FUNCTION_BLOCK CylControl (* Basic Function Block Type *)
  (* Standard: 61499-2 *)
  (* Version 0.0, 8/12/2014, valvya, nxtControl GmbH, Template *)
  PACKAGE Main;
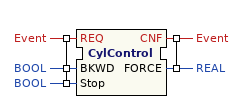
  EVENT_INPUT
    REQ WITH BKWD, Stop; (* Normal Execution Request *)
  END_EVENT
  EVENT_OUTPUT
    CNF WITH FORCE; (* Execution Confirmation *)
  END_EVENT
  VAR_INPUT
    BKWD : BOOL; (* Input event qualifier *)
    Stop : BOOL;
  END_VAR
  VAR_OUTPUT
    FORCE : REAL; (* Output event qualifier *)
  END_VAR
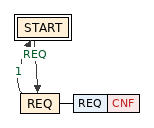
  EC_STATES
    START; (* Initial State *)
    REQ : REQ -> CNF; (* Normal execution *)
  END_STATES
  EC_TRANSITIONS
    START TO REQ := REQ;
    REQ TO START := 1;
  END_TRANSITIONS
  ALGORITHM REQ IN ST: (* Normally executed algorithm *)
IF BKWD AND NOT(Stop) THEN
  FORCE:=100;
ELSIF NOT(BKWD) AND Stop THEN
  FORCE :=0;
ELSE
	FORCE :=-100;
END_IF;
  END_ALGORITHM
END_FUNCTION_BLOCK
